PROGRAM PRG_Main_Chamber
VAR
END_VAR

(******************************************************************************************************)
(*Main Chamber*)
(******************************************************************************************************)
(*GAUGES*)
//Pirani Gauges
DREAM_MC_GPI_01.M_SetBits(30518);
DREAM_MC_GPI_01();

//Hot Cathode Guages
//DREAM_CAT1_GHC_01.M_SetBits(30518); //Not in the scope anymore
//DREAM_CAT1_GHC_01(PG:= DREAM_MC_GPI_01.PG); //Not in the scope anymore
DREAM_CAT2_GHC_01.M_SetBits(30518);
DREAM_CAT2_GHC_01(PG:= DREAM_MC_GPI_01.PG);
//Hot Cathode gauge IE514
DREAM_MC_GHC.M_SetBits(30518);
DREAM_MC_GHC(PG:= DREAM_MC_GPI_01.PG); //This fb reads statuses and control two gauges DREAM:MC:GHC:01 and DREAM:MC:GHC:02

(*VALVES*)
DREAM_CAT1_VRC_01(i_xExtILK_OK := FALSE, i_xOverrideMode := xSystemOverrideMode);

(*PUMPS*)
DREAM_MC_PTM_01(i_xExtIlkOK:= FALSE, iq_stPTM => );
DREAM_MC_PTM_02(i_xExtIlkOK:= FALSE, iq_stPTM => );

DREAM_CAT1_PTM_01(i_xExtIlkOK:= FALSE, iq_stPTM => );
DREAM_CAT2_PTM_01(i_xExtIlkOK:= FALSE, iq_stPTM => );

(*ROUGHING SECTION TURBO PUMPS*)
DREAM_ROUGH2_PTM_01(i_xExtIlkOK:= FALSE, iq_stPTM => );
DREAM_ROUGH2_PTM_02(i_xExtIlkOK:= FALSE, iq_stPTM => );

(******************************************************************************************************)
(*Serial Communication*)
(******************************************************************************************************)
//Leybold pumps
//DREAM_MC_PTM_01
(*Instanitate the Function block for serial communication with TD20 controller*)
fbTD20Com_DREAM_MC_PTM_01(SerialRXBuffer:= SerialRXBuffer_DREAM_MC_PTM_01,
                           SerialTXBuffer:= SerialTXBuffer_DREAM_MC_PTM_01,
                           astTD20Status=> stTD20_RBK_DREAM_MC_PTM_01);
(*Copy Status Pv's into the PTM structure*)
DREAM_MC_PTM_01.M_Serial_IO(stTD20_RBK_DREAM_MC_PTM_01);

//DREAM_MC_PTM_02
fbTD20Com_DREAM_MC_PTM_02(SerialRXBuffer:= SerialRXBuffer_DREAM_MC_PTM_02,
                           SerialTXBuffer:= SerialTXBuffer_DREAM_MC_PTM_02,
                           astTD20Status=> stTD20_RBK_DREAM_MC_PTM_02);

DREAM_MC_PTM_02.M_Serial_IO(stTD20_RBK_DREAM_MC_PTM_02);

//DREAM_CAT1_PTM_01 (TD400)
fbTD400Com_DREAM_CAT1_PTM_01(SerialRXBuffer:= SerialRXBuffer_DREAM_CAT1_PTM_01,
                             SerialTXBuffer:= SerialTXBuffer_DREAM_CAT1_PTM_01,
                             stTD400Control:= stTD400_CTRL_DREAM_CAT1_PTM_01,
                             stTD400Status=> stTD400_RBK_DREAM_CAT1_PTM_01);

//DREAM_CAT1_PTM_01.M_Serial_IO(stTD400_RBK_DREAM_CAT1_PTM_01);

//DREAM_CAT2_PTM_01 (TD400)
fbTD400Com_DREAM_CAT2_PTM_01(SerialRXBuffer:= SerialRXBuffer_DREAM_CAT2_PTM_01,
                             SerialTXBuffer:= SerialTXBuffer_DREAM_CAT2_PTM_01,
                             astTD20Status=> stTD400_RBK_DREAM_CAT2_PTM_01);

DREAM_CAT2_PTM_01.M_Serial_IO(stTD400_RBK_DREAM_CAT2_PTM_01);

//DREAM_ROUGH2_PTM_01 (TD400)
fbTD400Com_DREAM_ROUGH2_PTM_01(SerialRXBuffer:= SerialRXBuffer_DREAM_ROUGH2_PTM_01,
                               SerialTXBuffer:= SerialTXBuffer_DREAM_ROUGH2_PTM_01,
                               astTD20Status=> stTD400_RBK_DREAM_ROUGH2_PTM_01);

DREAM_ROUGH2_PTM_01.M_Serial_IO(stTD400_RBK_DREAM_ROUGH2_PTM_01);

//Pfeiffer pumps
//DREAM_NC_PTM_02 (Pfeiffer TC110)
stPfeiffer_CTRL_DREAM_ROUGH2_PTM_02[1].iSerialAddress:= 1;
stPfeiffer_CTRL_DREAM_ROUGH2_PTM_02[1].xEnableComm:= TRUE;
fbPfeifferCom_DREAM_ROUGH2_PTM_02(astPfeifferControl:= stPfeiffer_CTRL_DREAM_ROUGH2_PTM_02,
                                  astPfeifferStatus:= stPfeiffer_RBK_DREAM_ROUGH2_PTM_02,
                                  SerialRXBuffer:= SerialRXBuffer_DREAM_ROUGH2_PTM_02,
                                  SerialTXBuffer:= SerialTXBuffer_DREAM_ROUGH2_PTM_02);

DREAM_ROUGH2_PTM_02.M_Serial_IO(st_Pfeiffer_RBK:= stPfeiffer_RBK_DREAM_ROUGH2_PTM_02[1],
                                st_Pfeiffer_CTRL:= stPfeiffer_CTRL_DREAM_ROUGH2_PTM_02[1]);

END_PROGRAM

(* stored: Version 1.1.0.1, ProductVersion 3.1.4024.12
   POU PRG_Main_Chamber: Id {563898ad-99a3-4a88-bce1-94f471bfe1e1}, SpecialFunc None *)
